// TIA Portal project "MC" (V19)

(* hardware
DEVICE "S7-1200 station_1"  S7-1200 Station
   slot 0: "Rack_0"  S7-1200 Rack  Rack  V1.0
   slot 1: "PLC_1"  CPU 1212C DC/DC/Rly  6ES7 212-1HE40-0XB0  V4.6
*)

// ===== PLC "PLC_1"  CPU 1212C DC/DC/Rly =====

VAR_GLOBAL   // PLC tag table "Default tag table"
   "MotorSupply" AT %Q0.0 : Bool;
   "Start" AT %I0.0 : Bool;
   "Stop" AT %I0.1 : Bool;
   "Emergency" AT %I0.2 : Bool;
   "MotorOnLED" AT %Q0.1 : Bool;
   "MotorOffLED" AT %Q0.2 : Bool;
   "Motor2Supply" AT %Q0.3 : Bool;
   "ImpulsiStop" AT %I0.3 : Bool;
   "ImpulsiStart" AT %I0.4 : Bool;
   "AppoggioN1" AT %I0.5 : Bool;
   "Motor3Supply" AT %Q0.4 : Bool;
END_VAR

// folder: System blocks/Program resources

DATA_BLOCK "TP1"   // DB1
{ S7_Optimized_Access := 'TRUE' }
AUTHOR : Simatic
FAMILY : IEC
NAME : IEC_TMR
VERSION : 1.0
// stored: InstanceOfName IEC_TIMER
"IEC_TIMER"
BEGIN
END_DATA_BLOCK

DATA_BLOCK "TP2"   // DB2
{ S7_Optimized_Access := 'TRUE' }
AUTHOR : Simatic
FAMILY : IEC
NAME : IEC_TMR
VERSION : 1.0
// stored: InstanceOfName IEC_TIMER
"IEC_TIMER"
BEGIN
END_DATA_BLOCK

DATA_BLOCK "TP3"   // DB3
{ S7_Optimized_Access := 'TRUE' }
AUTHOR : Simatic
FAMILY : IEC
NAME : IEC_TMR
VERSION : 1.0
// stored: InstanceOfName IEC_TIMER
"IEC_TIMER"
BEGIN
END_DATA_BLOCK

DATA_BLOCK "TON1"   // DB4
{ S7_Optimized_Access := 'TRUE' }
AUTHOR : Simatic
FAMILY : IEC
NAME : IEC_TMR
VERSION : 1.0
// stored: InstanceOfName IEC_TIMER
"IEC_TIMER"
BEGIN
END_DATA_BLOCK

DATA_BLOCK "TON2"   // DB5
{ S7_Optimized_Access := 'TRUE' }
AUTHOR : Simatic
FAMILY : IEC
NAME : IEC_TMR
VERSION : 1.0
// stored: InstanceOfName IEC_TIMER
"IEC_TIMER"
BEGIN
END_DATA_BLOCK

DATA_BLOCK "TON3"   // DB6
{ S7_Optimized_Access := 'TRUE' }
AUTHOR : Simatic
FAMILY : IEC
NAME : IEC_TMR
VERSION : 1.0
// stored: InstanceOfName IEC_TIMER
"IEC_TIMER"
BEGIN
END_DATA_BLOCK

DATA_BLOCK "TP4"   // DB7
{ S7_Optimized_Access := 'TRUE' }
AUTHOR : Simatic
FAMILY : IEC
NAME : IEC_TMR
VERSION : 1.0
// stored: InstanceOfName IEC_TIMER
"IEC_TIMER"
BEGIN
END_DATA_BLOCK

DATA_BLOCK "CU1"   // DB8
{ S7_Optimized_Access := 'TRUE' }
AUTHOR : Simatic
FAMILY : IEC
NAME : CNTR
VERSION : 1.0
// stored: InstanceOfName IEC_COUNTER
"IEC_COUNTER"
BEGIN
END_DATA_BLOCK

DATA_BLOCK "TONR1"   // DB9
{ S7_Optimized_Access := 'TRUE' }
AUTHOR : Simatic
FAMILY : IEC
NAME : IEC_TMR
VERSION : 1.0
// stored: InstanceOfName IEC_TIMER
"IEC_TIMER"
BEGIN
END_DATA_BLOCK

// folder: (top level)

ORGANIZATION_BLOCK "Main"   // OB1, LAD, ProgramCycle
TITLE = "Main Program Sweep (Cycle)"
{ S7_Optimized_Access := 'TRUE' }
VERSION : 0.1
   VAR_INPUT
      Initial_Call : Bool;   // Initial call of this OB
      Remanence : Bool;   // =True, if remanent data are available
   END_VAR
   VAR_TEMP   // added for the SCL form of the ladder/FBD networks
      _w1 : Bool;
   END_VAR
BEGIN

REGION Network 1
   // Autoritenuta bobina normale
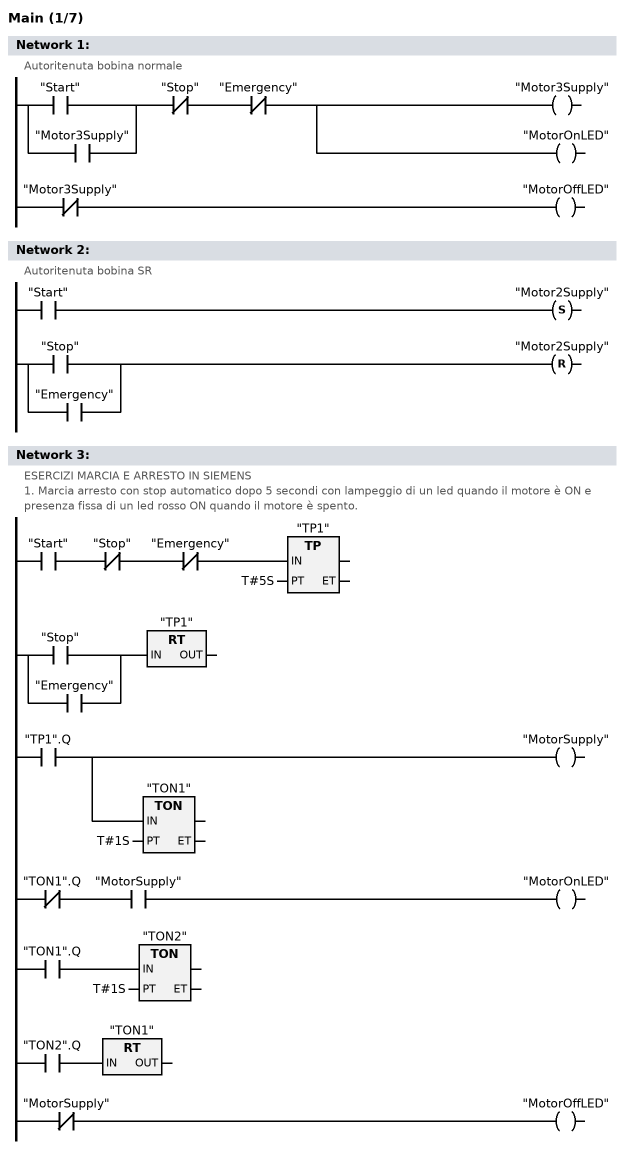
   RUNG wire#powerrail
      Contact( "Start" )
      wire#w1
      I_Contact( "Stop" )
      I_Contact( "Emergency" )
      wire#w2
      Coil( "Motor3Supply" )
   END_RUNG
   RUNG wire#powerrail
      Contact( "Motor3Supply" )
   END_RUNG wire#w1
   RUNG wire#w2
      Coil( "MotorOnLED" )
   END_RUNG
   RUNG wire#powerrail
      I_Contact( "Motor3Supply" )
      Coil( "MotorOffLED" )
   END_RUNG
   // the same network as SCL:
   "Motor3Supply" := ("Start" OR "Motor3Supply") AND NOT "Stop" AND NOT "Emergency";
   "MotorOnLED" := "Motor3Supply";
   "MotorOffLED" := NOT "Motor3Supply";
END_REGION

REGION Network 2
   // Autoritenuta bobina SR
   RUNG wire#powerrail
      Contact( "Start" )
      S_Coil( "Motor2Supply" )
   END_RUNG
   RUNG wire#powerrail
      Contact( "Stop" )
      wire#w1
      R_Coil( "Motor2Supply" )
   END_RUNG
   RUNG wire#powerrail
      Contact( "Emergency" )
   END_RUNG wire#w1
   // the same network as SCL:
   IF "Start" THEN "Motor2Supply" := TRUE; END_IF;
   IF "Stop" OR "Emergency" THEN "Motor2Supply" := FALSE; END_IF;
END_REGION

REGION Network 3
   // ESERCIZI MARCIA E ARRESTO IN SIEMENS
   // 
   // 1. Marcia arresto con stop automatico dopo 5 secondi con lampeggio di un led quando il motore è ON e presenza fissa di un led rosso ON quando il motore è spento.
   "TP1".TP(IN := "Start" AND NOT "Stop" AND NOT "Emergency", PT := T#5S);
   IF "Stop" OR "Emergency" THEN RESET_TIMER("TP1"); END_IF;
   "MotorSupply" := "TP1".Q;
   "TON1".TON(IN := "TP1".Q, PT := T#1S);
   "MotorOnLED" := NOT "TON1".Q AND "MotorSupply";
   "TON2".TON(IN := "TON1".Q, PT := T#1S);
   IF "TON2".Q THEN RESET_TIMER("TON1"); END_IF;
   "MotorOffLED" := NOT "MotorSupply";
END_REGION

REGION Network 4
   // Alternativa: 2 TP autoescludenti
   // 
   // TP2 va resettato forzatamente quando il motore si spegne perchè potrebbe essere ancora eccitato quando ciò accade
   // 
   // NOTA: TP2 viene alimentato prima di TP3 per ordine di esecuzione del programma
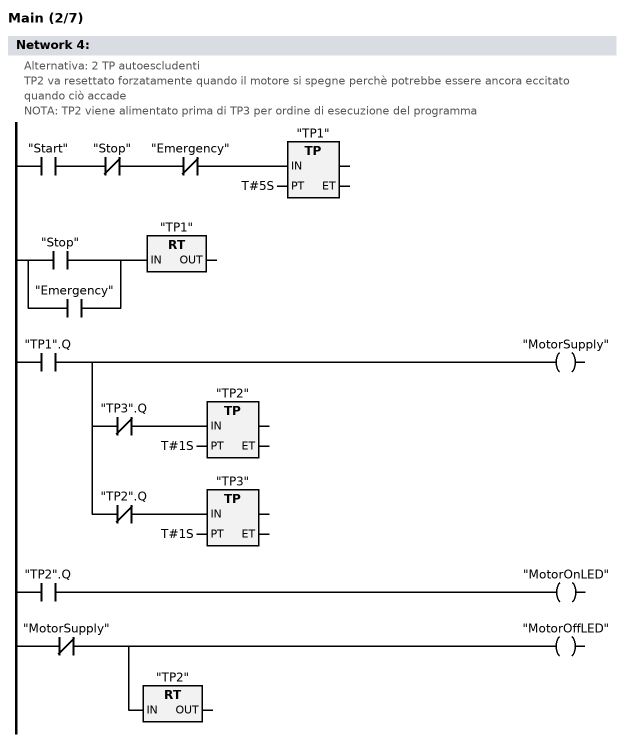
   "TP1".TP(IN := "Start" AND NOT "Stop" AND NOT "Emergency", PT := T#5S);
   IF "Stop" OR "Emergency" THEN RESET_TIMER("TP1"); END_IF;
   "MotorSupply" := "TP1".Q;
   "TP2".TP(IN := "TP1".Q AND NOT "TP3".Q, PT := T#1S);
   "TP3".TP(IN := "TP1".Q AND NOT "TP2".Q, PT := T#1S);
   "MotorOnLED" := "TP2".Q;
   "MotorOffLED" := NOT "MotorSupply";
   IF NOT "MotorSupply" THEN RESET_TIMER("TP2"); END_IF;
END_REGION

REGION Network 5
   // 2. Marcia arresto con partenza ritardata dopo 5 secondi, con lampeggio di un led quando il motore è ON, in cui 1 S è acceso e 2 S è spento, e presenza fissa di un led rosso ON quando il motore è spento.
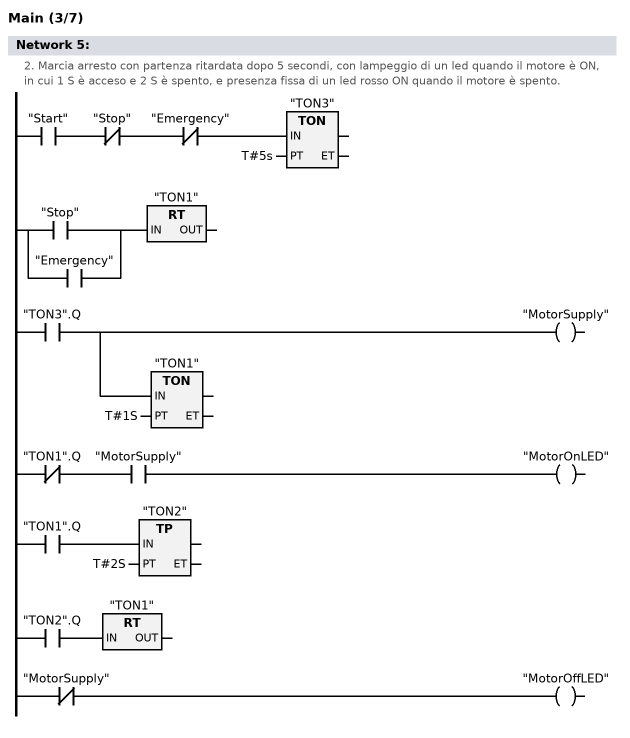
   "TON3".TON(IN := "Start" AND NOT "Stop" AND NOT "Emergency", PT := T#5s);
   IF "Stop" OR "Emergency" THEN RESET_TIMER("TON1"); END_IF;
   "MotorSupply" := "TON3".Q;
   "TON1".TON(IN := "TON3".Q, PT := T#1S);
   "MotorOnLED" := NOT "TON1".Q AND "MotorSupply";
   "TON2".TP(IN := "TON1".Q, PT := T#2S);
   IF "TON2".Q THEN RESET_TIMER("TON1"); END_IF;
   "MotorOffLED" := NOT "MotorSupply";
END_REGION

REGION Network 6
   // 3. Marcia arresto con partenza ritardata dopo 5 secondi e stop automatico dopo 5 secondi con lampeggio di un led quando il motore è ON in cui 1 S è acceso e 2 S è spento e presenza fissa di un led rosso ON quando il motore è spento.
   // 
   // NOTA: si può usare TP con rilevamente fronte discesa Q per azionare/spegnere il motore dopo scorrimento 5s di TP (e non quando Q è a zero prima dell'eccitamento..)
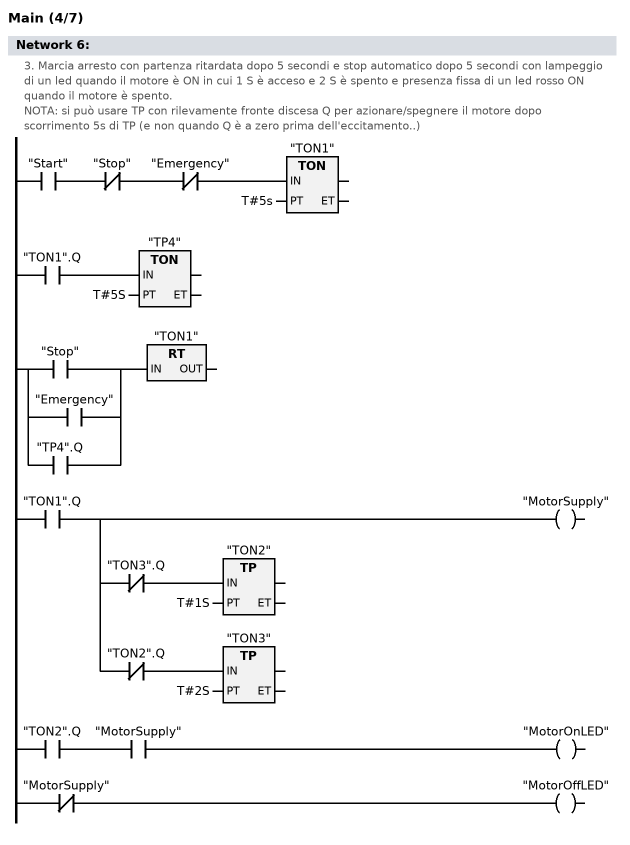
   "TON1".TON(IN := "Start" AND NOT "Stop" AND NOT "Emergency", PT := T#5s);
   "TP4".TON(IN := "TON1".Q, PT := T#5S);
   IF "Stop" OR "Emergency" OR "TP4".Q THEN RESET_TIMER("TON1"); END_IF;
   "MotorSupply" := "TON1".Q;
   "TON2".TP(IN := "TON1".Q AND NOT "TON3".Q, PT := T#1S);
   "TON3".TP(IN := "TON1".Q AND NOT "TON2".Q, PT := T#2S);
   "MotorOnLED" := "TON2".Q AND "MotorSupply";
   "MotorOffLED" := NOT "MotorSupply";
END_REGION

REGION Network 7
   // 4. Marcia arresto con stop automatico dopo 5 impulsi su I3 con lampeggio di un led quando il motore è ON in cui 1 S è acceso e 2 S è spento e presenza fissa di un led rosso ON quando il motore è spento.
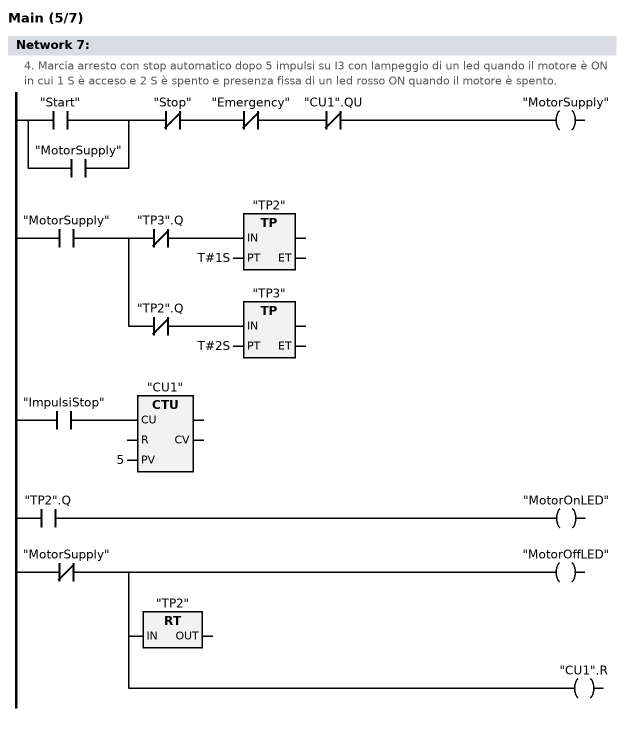
   "MotorSupply" := ("Start" OR "MotorSupply") AND NOT "Stop" AND NOT "Emergency" AND NOT "CU1".QU;
   "TP2".TP(IN := "MotorSupply" AND NOT "TP3".Q, PT := T#1S);
   "TP3".TP(IN := "MotorSupply" AND NOT "TP2".Q, PT := T#2S);
   "CU1".CTU(CU := "ImpulsiStop", PV := 5);
   "MotorOnLED" := "TP2".Q;
   "MotorOffLED" := NOT "MotorSupply";
   IF NOT "MotorSupply" THEN RESET_TIMER("TP2"); END_IF;
   "CU1".R := NOT "MotorSupply";
END_REGION

REGION Network 8
   // 5. Marcia arresto con partenza ritardata dopo 5 impulsi su I3 oppure premendo marcia fisico, con lampeggio di un led quando il motore è ON in cui 1 S è acceso e 2 S è spento e presenza fissa di un led rosso ON quando il motore è spento.
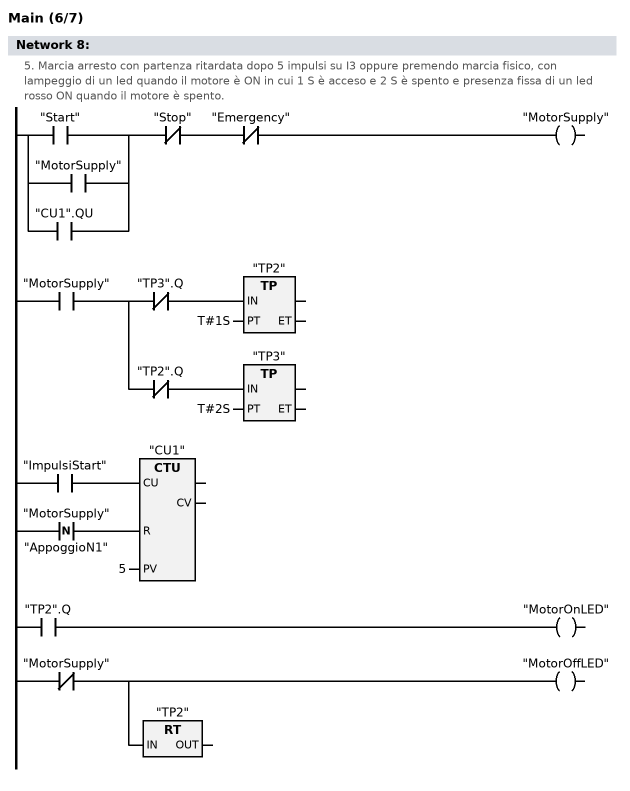
   "MotorSupply" := ("Start" OR "MotorSupply" OR "CU1".QU) AND NOT "Stop" AND NOT "Emergency";
   "TP2".TP(IN := "MotorSupply" AND NOT "TP3".Q, PT := T#1S);
   "TP3".TP(IN := "MotorSupply" AND NOT "TP2".Q, PT := T#2S);
   #_w1 := NOT "MotorSupply" AND "AppoggioN1";   // falling edge of "MotorSupply"
   "AppoggioN1" := "MotorSupply";
   "CU1".CTU(CU := "ImpulsiStart", R := #_w1, PV := 5);
   "MotorOnLED" := "TP2".Q;
   "MotorOffLED" := NOT "MotorSupply";
   IF NOT "MotorSupply" THEN RESET_TIMER("TP2"); END_IF;
END_REGION

REGION Network 9
   // 6. Marcia arresto di un motore che si avvii dopo che la marcia è stata tenuta premuta (anche in momenti diversi) per un totale di 25 s, con lampeggio di un led quando il motore è ON in cui 1 S è acceso e 2 S è spento e presenza fissa di un led rosso ON quando il motore è spento.
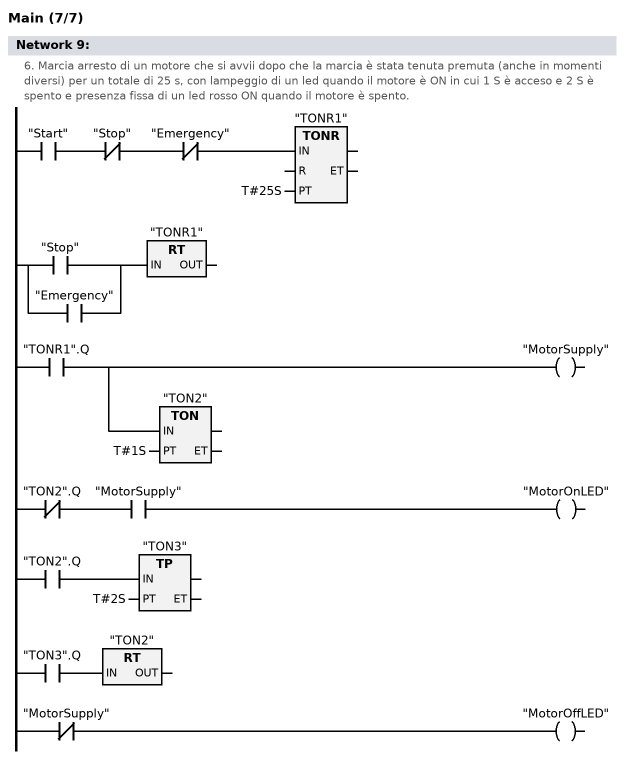
   "TONR1".TONR(IN := "Start" AND NOT "Stop" AND NOT "Emergency", PT := T#25S);
   IF "Stop" OR "Emergency" THEN RESET_TIMER("TONR1"); END_IF;
   "MotorSupply" := "TONR1".Q;
   "TON2".TON(IN := "TONR1".Q, PT := T#1S);
   "MotorOnLED" := NOT "TON2".Q AND "MotorSupply";
   "TON3".TP(IN := "TON2".Q, PT := T#2S);
   IF "TON3".Q THEN RESET_TIMER("TON2"); END_IF;
   "MotorOffLED" := NOT "MotorSupply";
END_REGION
END_ORGANIZATION_BLOCK